(* PLC project KinIn_v3.project, CODESYS CODESYS V3.5 SP19 *)
(* stored: creationDateTime 2025-01-20T16:22:07.2595442, modificationDateTime 2025-01-20T16:17:39.6822999 *)

FUNCTION_BLOCK LuDecomposition
  VAR_INPUT
    {attribute 'variable_length_array_original_scope' := 'Inout'}
    {attribute 'variable_length_array' := 'ARRAY[*,*] OF REAL'}
    {attribute 'Dimensions' := '2'}
    A : POINTER TO REAL;
    {attribute 'variable_length_array_original_scope' := 'Inout'}
    {attribute 'variable_length_array' := 'ARRAY[*,*] OF REAL'}
    {attribute 'Dimensions' := '2'}
    L : POINTER TO REAL;
    {attribute 'variable_length_array_original_scope' := 'Inout'}
    {attribute 'variable_length_array' := 'ARRAY[*,*] OF REAL'}
    {attribute 'Dimensions' := '2'}
    U : POINTER TO REAL;
  END_VAR
  VAR
    i : DINT;
    j : DINT;
    k : DINT;
    u_SumTemp : REAL;  (* using temporal variables for more clarity *)
    l_SumTemp : REAL;
  END_VAR

            //initialize both arrays as 0
i:=1;j:=1;
FOR i:=1 TO UPPER_BOUND(L,1) DO
	FOR j:=1 TO UPPER_BOUND(L,2) DO
		L[i,j]:=0;
		U[i,j]:=0;
	END_FOR
END_FOR

i:=1;j:=1;
FOR i:=1 TO UPPER_BOUND(L,1) DO
	FOR j:=1 TO UPPER_BOUND(L,2) DO
		
	//j only oparates when is greater or equal than 1
		IF (j>=i) THEN
			u_SumTemp:=0;k:=1;
			FOR k:=1 TO i-1 DO
				u_SumTemp:=u_SumTemp+L[i,k]*U[k,j];
			END_FOR
			U[i,j]:=A[i,j]-u_SumTemp;//the complex formula for it
			
			IF j=i THEN
				L[j,i]:=1;
			ELSE //(j<>i)
				l_SumTemp:=0;k:=1;
				FOR k:=1 TO i-1 DO
					l_SumTemp:=l_SumTemp+L[j,k]*U[k,i];
				END_FOR
				//the complex formula
				IF U[i,i]=0 AND (A[j,i]-l_SumTemp)=0 THEN
					L[j,i]:=1;
				ELSIF U[i,i]=0 THEN
					L[j,i]:=3.402823E+10;
				ELSE
					L[j,i]:=(A[j,i]-l_SumTemp)/U[i,i];//the complex formula
				END_IF
		

			END_IF
		END_IF
	//the rest of values are zeros
	END_FOR
END_FOR
          
END_FUNCTION_BLOCK
